TYPE INTERNAL  _BroadcastUnion :
UNION
	iSignal		: I_SignalNode;
	iReceiver	: I_ReceiverNode;
END_UNION
END_TYPE

(* stored: Version 1.1.0.1
   DUT _BroadcastUnion: Id {5c7e35f6-1446-412c-affd-6d2f069720fe} *)
